{attribute 'qualified_only'}
{attribute 'strict'}
TYPE
    eDialogAnswer :
    (
        NoAnswer := 0,
        OK       := 10,
        Yes      := 20,
        No       := 30,
        Cancel   := 40,
		Invoked	  :=50
    );
END_TYPE

(* stored: Version 1.1.0.1
   DUT eDialogAnswer: Id {ad0c95f8-cac1-07f0-37b4-7e14b4b70031} *)
